INTERFACE I_Logger

METHOD M_WriteData : Bool

VAR_INPUT
	execute : BOOL;         // Trigger for logging
	data : STRING;
END_VAR
END_METHOD

END_INTERFACE

(* stored: Version 1.1.0.1
   Itf I_Logger: Id {a2cc0595-dcf5-4a2c-a6d6-5db81b8f9948}
   Method M_WriteData: Id {691a339b-cc79-4aca-9400-312c622d5676} *)
